// Mitsubishi GX Works2 project: 타이머_카운터응용   PLC: Q02/Q02H

PROGRAM MAIN
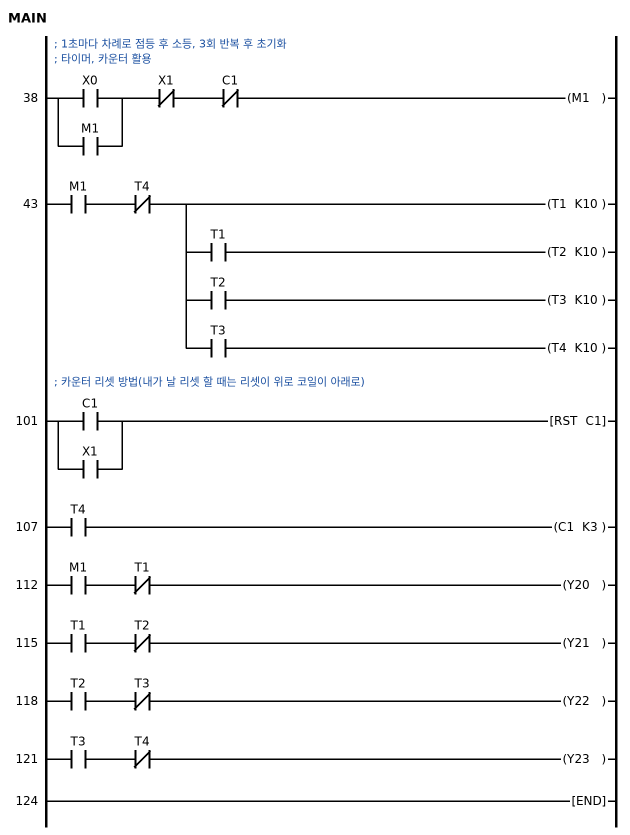
; 1초마다 차례로 점등 후 소등, 3회 반복 후 초기화
; 타이머, 카운터 활용
38    LD      X0
      OR      M1
      ANI     X1
      ANI     C1
      OUT     M1
43    LD      M1
      ANI     T4
      OUT     T1 K10
      MPS
      AND     T1
      OUT     T2 K10
      MRD
      AND     T2
      OUT     T3 K10
      MPP
      AND     T3
      OUT     T4 K10
; 카운터 리셋 방법(내가 날 리셋 할 때는 리셋이 위로 코일이 아래로)
101   LD      C1
      OR      X1
      RST     C1
107   LD      T4
      OUT     C1 K3
112   LD      M1
      ANI     T1
      OUT     Y20
115   LD      T1
      ANI     T2
      OUT     Y21
118   LD      T2
      ANI     T3
      OUT     Y22
121   LD      T3
      ANI     T4
      OUT     Y23
124   END
END_PROGRAM
